SYSTEM Simple2mon
  (* Version 1.0, 2019-11-01, badger *)
  APPLICATION Simple2monApp
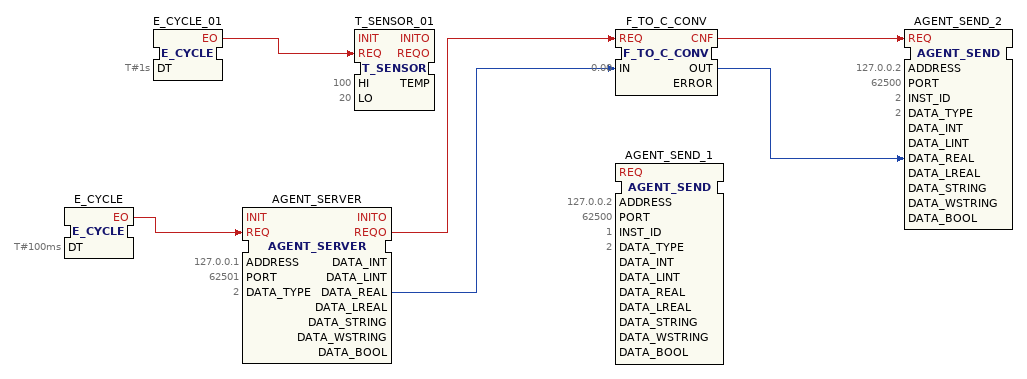
    FBS
      E_CYCLE_01 : E_CYCLE(DT := T#1s);
      T_SENSOR_01 : T_SENSOR(HI := 100, LO := 20);
      AGENT_SERVER : AGENT_SERVER(ADDRESS := 127.0.0.1, PORT := 62501, DATA_TYPE := 2);
      E_CYCLE : E_CYCLE(DT := T#100ms);
      AGENT_SEND_2 : AGENT_SEND(ADDRESS := 127.0.0.2, PORT := 62500, INST_ID := 2, DATA_TYPE := 2);
      F_TO_C_CONV : F_TO_C_CONV(IN := 0.00);
      AGENT_SEND_1 : AGENT_SEND(ADDRESS := 127.0.0.2, PORT := 62500, INST_ID := 1, DATA_TYPE := 2);
    END_FBS
    EVENT_CONNECTIONS
      E_CYCLE_01.EO TO T_SENSOR_01.REQ;
      F_TO_C_CONV.CNF TO AGENT_SEND_2.REQ;
      E_CYCLE.EO TO AGENT_SERVER.REQ;
      AGENT_SERVER.REQO TO F_TO_C_CONV.REQ;
    END_CONNECTIONS
    DATA_CONNECTIONS
      F_TO_C_CONV.OUT TO AGENT_SEND_2.DATA_REAL;
      AGENT_SERVER.DATA_REAL TO F_TO_C_CONV.IN;
    END_CONNECTIONS
  END_APPLICATION
  DEVICE FORTE_PC : FORTE_PC(MGR_ID := "localhost:61499")
    {SET_ATTRIBUTE(Profile, HOLOBLOC)} (* device profile *)
    RESOURCE EMB_RES : EMB_RES
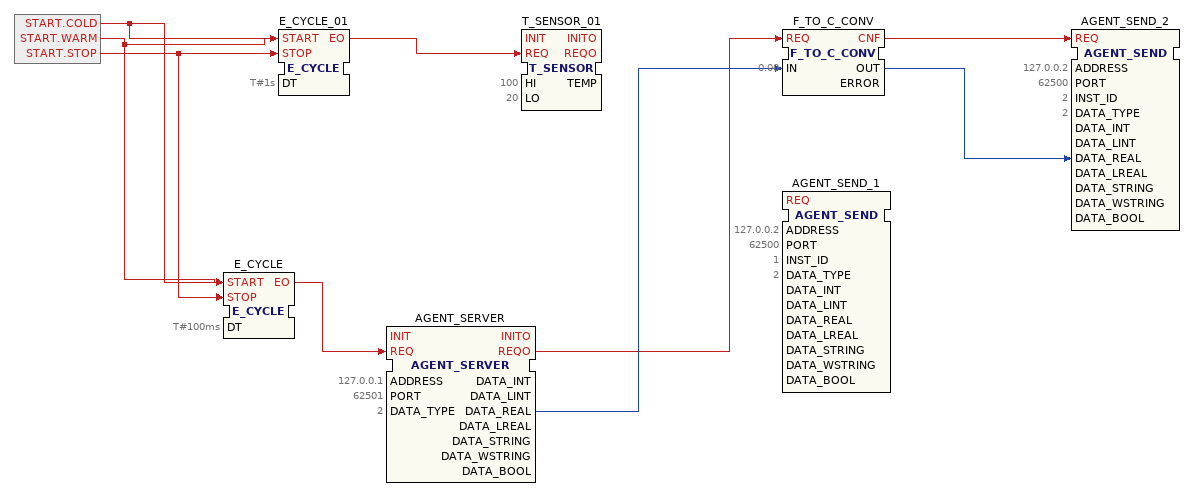
      FBS
        E_CYCLE_01 : E_CYCLE(DT := T#1s);
        E_CYCLE : E_CYCLE(DT := T#100ms);
        AGENT_SERVER : AGENT_SERVER(ADDRESS := 127.0.0.1, PORT := 62501, DATA_TYPE := 2);
        F_TO_C_CONV : F_TO_C_CONV(IN := 0.00);
        AGENT_SEND_1 : AGENT_SEND(ADDRESS := 127.0.0.2, PORT := 62500, INST_ID := 1, DATA_TYPE := 2);
        AGENT_SEND_2 : AGENT_SEND(ADDRESS := 127.0.0.2, PORT := 62500, INST_ID := 2, DATA_TYPE := 2);
        T_SENSOR_01 : T_SENSOR(HI := 100, LO := 20);
      END_FBS
      EVENT_CONNECTIONS
        F_TO_C_CONV.CNF TO AGENT_SEND_2.REQ;
        E_CYCLE_01.EO TO T_SENSOR_01.REQ;
        START.COLD TO E_CYCLE_01.START;
        START.WARM TO E_CYCLE_01.START;
        START.STOP TO E_CYCLE_01.STOP;
        E_CYCLE.EO TO AGENT_SERVER.REQ;
        AGENT_SERVER.REQO TO F_TO_C_CONV.REQ;
        START.COLD TO E_CYCLE.START;
        START.WARM TO E_CYCLE.START;
        START.STOP TO E_CYCLE.STOP;
      END_CONNECTIONS
      DATA_CONNECTIONS
        F_TO_C_CONV.OUT TO AGENT_SEND_2.DATA_REAL;
        AGENT_SERVER.DATA_REAL TO F_TO_C_CONV.IN;
      END_CONNECTIONS
    END_RESOURCE
  END_DEVICE
  MAPPINGS
    Simple2monApp.E_CYCLE_01 ON FORTE_PC.EMB_RES.E_CYCLE_01;
    Simple2monApp.E_CYCLE ON FORTE_PC.EMB_RES.E_CYCLE;
    Simple2monApp.AGENT_SERVER ON FORTE_PC.EMB_RES.AGENT_SERVER;
    Simple2monApp.F_TO_C_CONV ON FORTE_PC.EMB_RES.F_TO_C_CONV;
    Simple2monApp.AGENT_SEND_1 ON FORTE_PC.EMB_RES.AGENT_SEND_1;
    Simple2monApp.AGENT_SEND_2 ON FORTE_PC.EMB_RES.AGENT_SEND_2;
    Simple2monApp.T_SENSOR_01 ON FORTE_PC.EMB_RES.T_SENSOR_01;
  END_MAPPINGS
  SEGMENTS
    Ethernet : Ethernet;
  END_SEGMENTS
  LINKS
    FORTE_PC => Ethernet;
  END_LINKS
END_SYSTEM
